{attribute 'GeneratedUsingTerminal: EPP3314-0002-0016'}
{attribute addProperty BoxType "EPP3314-0002-0016"}
{attribute addProperty Id "EtcSlaveTerminalBaseTC_Inputs_Channel_1AT %I*TC_Inputs_Channel_4A3944819TC_Inputs_Channel_2AT %I*TC_Inputs_Channel_4A3944819TC_Inputs_Channel_3AT %I*TC_Inputs_Channel_4A3944819TC_Inputs_Channel_4AT %I*TC_Inputs_Channel_4A3944819WcStateAT %I*WcState_9091E0EB2InfoDataAT %I*InfoData_32EB74EA10"}
{attribute addProperty CRC "1811037525"}
{attribute addProperty Size "48"}
TYPE EPP3314_6BF23D55 EXTENDS EtcSlaveTerminalBase :
STRUCT
	{attribute addProperty Name "TC_Inputs_Channel_1"}
	TC_Inputs_Channel_1 : TC_Inputs_Channel_4A394481;
	{attribute addProperty Name "TC_Inputs_Channel_2"}
	TC_Inputs_Channel_2 : TC_Inputs_Channel_4A394481;
	{attribute addProperty Name "TC_Inputs_Channel_3"}
	TC_Inputs_Channel_3 : TC_Inputs_Channel_4A394481;
	{attribute addProperty Name "TC_Inputs_Channel_4"}
	TC_Inputs_Channel_4 : TC_Inputs_Channel_4A394481;
	{attribute addProperty Name "WcState"}
	WcState : WcState_9091E0EB;
	{attribute addProperty Name "InfoData"}
	InfoData : InfoData_32EB74EA;
END_STRUCT
END_TYPE

(* stored: Version 1.2.0.0, ProductVersion 3.1.4024.9
   DUT EPP3314_6BF23D55: Id {459e9bca-0ad6-4de4-b1df-c34ba37c5345} *)
